FUNCTION_BLOCK trip_pulse_timer (* Basic Function Block Type *)
  (* Standard: 61499-2 *)
  (* Version 0.0, 11/29/2016, gulzha, nxtControl GmbH, Template *)
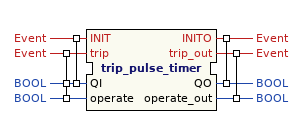
  EVENT_INPUT
    INIT WITH QI; (* Initialization Request *)
    trip WITH QI, operate; (* Normal Execution Request *)
  END_EVENT
  EVENT_OUTPUT
    INITO WITH QO; (* Initialization Confirm *)
    trip_out WITH operate_out;
  END_EVENT
  VAR_INPUT
    QI : BOOL; (* Input event qualifier *)
    operate : BOOL;
  END_VAR
  VAR_OUTPUT
    QO : BOOL; (* Output event qualifier *)
    operate_out : BOOL;
  END_VAR
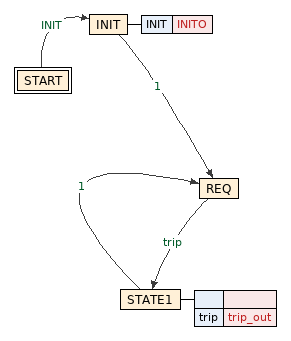
  EC_STATES
    START; (* Initial State *)
    INIT : INIT -> INITO; (* Initialization *)
    REQ; (* Normal execution *)
    STATE1 : trip -> trip_out;
  END_STATES
  EC_TRANSITIONS
    START TO INIT := INIT;
    INIT TO REQ := 1;
    REQ TO STATE1 := trip;
    STATE1 TO REQ := 1;
  END_TRANSITIONS
  ALGORITHM INIT IN ST: (* Initialization algorithm *)
;

operate := FALSE;
operate_out := FALSE;
  END_ALGORITHM
  ALGORITHM REQ IN ST: (* Normally executed algorithm *)
;
  END_ALGORITHM
  ALGORITHM trip IN ST:
;
operate_out := operate;
  END_ALGORITHM
  ALGORITHM reset IN ST:
;
operate_out := FALSE;
  END_ALGORITHM
END_FUNCTION_BLOCK
